// TIA Portal V19 export
VAR_GLOBAL   // PLC tag table "Em1"
END_VAR
